FUNCTION FUN_GetDate : STRING
VAR_INPUT
	stNtTime		:TIMESTRUCT;
END_VAR
VAR
	sDate			:STRING;
END_VAR

// Initialize string
sDate := '';

// Add year to string
sDate := UINT_TO_STRING(stNtTime.wYear);
sDate := CONCAT(sDate,'-');

// Add month to string
IF stNtTime.wMonth < 10 THEN
	sDate := CONCAT(sDate,'0');
END_IF
sDate := CONCAT(sDate,UINT_TO_STRING(stNtTime.wMonth));
sDate := CONCAT(sDate,'-');

// Add day to string
IF stNtTime.wDay < 10 THEN
	sDate := CONCAT(sDate, '0');
END_IF
sDate := CONCAT(sDate,UINT_TO_STRING(stNtTime.wDay));

// Return result
FUN_GetDate := sDate;

END_FUNCTION

(* stored: Version 1.1.0.1, ProductVersion 3.1.4024.12
   POU FUN_GetDate: Id {eabe7852-f754-4cbd-8df6-106a78b59095}, SpecialFunc None *)
